PROGRAM MAIN
VAR
	SinusValue :	REAL := 0;
	SquareValue:	REAL := 0;
	PWMValue:		REAL := 0;
	t:				REAL := 0;
END_VAR

SinusValue := SinusFunction(A:=2,yoff:=0,w:=2,t:=t);
SquareValue := SquareSignal(ymin:= 4, ymax := 3, w:= 5, yoff:= -1, t:=t);
PWMValue := PwmSignal(ymin:= 4, ymax := 3, w:= 5, yoff:= -1, t:=t, PWM:= 0.7);

t := t + 0.01;

END_PROGRAM

(* stored: Version 1.1.0.1, ProductVersion 3.1.4024.13
   POU MAIN: Id {aa14506c-e177-4d89-94bf-b04e2e20aa7f}, SpecialFunc None *)
